TEXTLIST RackText
  1 = 'Type1: "Long Straight"'
  2 = 'Type2: "Curved"'
  3 = 'Type3:  "Incline"'
  4 = 'Type4: "Decline"'
  5 = 'EL2008'
  6 = 'EL1008'
  7 = 'N/A'
  11 = 'Conveyer Type1: Long Straight: Ids 1-10'
  8 = 'Conveyer Type2: Curved: Ids 11-20'
  9 = 'Conveyer Type3: Incline: Ids 21-30'
  10 = 'Conveyer Type4: Decline: Ids 31-40'
  0 = ''
   = ''
END_TEXTLIST

(* stored: Version 1.1.0.1, ProductVersion 3.1.4024.6
   TextList RackText: Id {c967b551-e547-4604-bcdb-2721183a2370} *)
